{attribute 'linkalways'} 
{attribute 'no_explicit_call' := 'This FB is a CLASS and must be accessed using methods or properties'}
{attribute 'enable_dynamic_creation'}
FUNCTION_BLOCK FINAL ABS_USINT EXTENDS Node
VAR
	in : _USINT(0);
	out : _USINT(0);
END_VAR

METHOD PUBLIC Clone : I_Node
VAR
	pNode : POINTER TO ABS_USINT;
END_VAR
pNode := __NEW(ABS_USINT);
Clone := pNode^;
END_METHOD

METHOD FB_init : BOOL
VAR_INPUT
	bInitRetains : BOOL; // if TRUE, the retain variables are initialized (warm start / cold start)
	bInCopyCode : BOOL;  // if TRUE, the instance afterwards gets moved into the copy code (online change)
END_VAR
AddInput('in',THIS^.in);
AddOutput('out', THIS^.out);
END_METHOD

METHOD PROTECTED OnExecute
VAR
END_VAR
out.Value := ABS(in.Value);
END_METHOD

END_FUNCTION_BLOCK

(* stored: Version 1.1.0.1, ProductVersion 3.1.4024.15
   POU ABS_USINT: Id {4e81af29-38d8-4cde-9891-e22300ada466}, SpecialFunc None
   Folder Constructor: Id {a4381474-2a9f-4f9b-afbc-1650fbbe4798}
   Method Clone: Id {691810fe-4c0f-4b9b-9e59-a49244e1a6b0}
   Method FB_init: Id {6b4229f8-68a3-4ef6-808d-d919ecffa161}
   Method OnExecute: Id {d23ad1d2-0f87-4167-8201-9a7f15214d6d} *)
